(* CoDeSys 2.3.9.41 project: Lab4.pro *)
(* Libraries: STANDARD.LIB 5.6.98 11:03:02 *)

(* Task configuration *)
TASK Standard (PRIORITY := 0, INTERVAL := T#5ms);
	MAIN
END_TASK

(* Global variable list: Global_Variables *)
VAR_GLOBAL
END_VAR

VAR_GLOBAL CONSTANT
	F_TASK : INT := 200;
	PERIOD_TASK : INT := 5;
END_VAR

(* POU MAIN, ST *)
PROGRAM MAIN
VAR
	lp : LowpassFilter;
	integrate : Integrator;

END_VAR
Generator();
END_PROGRAM

(* POU LowpassFilter, ST *)
FUNCTION_BLOCK LowpassFilter
VAR_INPUT
	input : REAL;
	tau : INT;
END_VAR
VAR_OUTPUT
	output : REAL;
END_VAR
VAR
	sum : REAL := 0;
END_VAR
sum := (input * PERIOD_TASK + sum * tau) / (PERIOD_TASK + tau);
output := sum;
END_FUNCTION_BLOCK

(* POU Integrator, ST *)
FUNCTION_BLOCK Integrator
VAR_INPUT
	input : REAL;
END_VAR
VAR_OUTPUT
	output : REAL;
END_VAR
VAR
	sum : REAL := 0;
END_VAR
sum := sum + input;
output := sum;
END_FUNCTION_BLOCK

(* POU Generator, ST *)
PROGRAM Generator
VAR
	t : UINT := 0;
	a : REAL := 1;
	offset : REAL := 0;
	w : REAL := 1.0;
	duty : REAL := 0.25;
	sinus : REAL;
	square : REAL;
	pwm : REAL;
END_VAR
IF t <= REAL_TO_INT(w*F_TASK) THEN
	t := t + 1;
ELSE
	t := 0;
END_IF
sinus := SinusFunction(a, offset, w, t);
square := SquareSignal(a, offset, w, t);
pwm := PwmSignal(a, offset, w, t, duty);
END_PROGRAM

(* POU SinusFunction, ST *)
FUNCTION SinusFunction : REAL
VAR_INPUT
	a : REAL;
	offset : REAL;
	w : REAL;
	t : INT;
END_VAR
VAR
END_VAR
SinusFunction := a * SIN(INT_TO_REAL(t)*w /F_TASK *2.0*3.1415) + offset;
END_FUNCTION

(* POU SquareSignal, ST *)
FUNCTION SquareSignal : REAL
VAR_INPUT
	a : REAL;
	offset : REAL;
	w : REAL;
	t : INT;
END_VAR
VAR
	per : INT;
END_VAR
per := REAL_TO_INT(F_TASK / w);
IF (t MOD per) < (per / 2) THEN
	SquareSignal := offset + a;
ELSE
	SquareSignal := offset - a;
END_IF
END_FUNCTION

(* POU PwmSignal, ST *)
FUNCTION PwmSignal : REAL
VAR_INPUT
	a : REAL;
	offset : REAL;
	w : REAL;
	t : INT;
	duty : REAL;
END_VAR
VAR
	per : INT;
END_VAR
per := REAL_TO_INT(F_TASK / w);
IF duty*per >= per THEN
	PwmSignal := offset + a;
ELSIF duty*per <=0 THEN
	PwmSignal := offset - a;
ELSIF (t MOD per) < duty*per THEN
	PwmSignal := offset + a;
ELSE
	PwmSignal := offset - a;
END_IF
END_FUNCTION

(* POU EdgeDetector, ST *)
FUNCTION_BLOCK EdgeDetector
VAR_INPUT
	inputValue : BOOL;
END_VAR
VAR_OUTPUT
	risingEdge : BOOL;
	fallingEdge : BOOL;
END_VAR
VAR
	prev : BOOL := FALSE;
END_VAR
IF inputValue > prev THEN
	risingEdge := TRUE;
	fallingEdge := FALSE;
ELSIF inputValue < prev THEN
	risingEdge := FALSE;
	fallingEdge := TRUE;
ELSE
	risingEdge := FALSE;
	fallingEdge := FALSE;
END_IF
prev := inputValue;
END_FUNCTION_BLOCK

(* POU EdgeDetectorDouble, ST *)
FUNCTION_BLOCK EdgeDetectorDouble
VAR_INPUT
	inputValue : BOOL;
	threshold : INT;
END_VAR
VAR_OUTPUT
	risingEdge : BOOL;
	fallingEdge : BOOL;
	double : BOOL;
END_VAR
VAR
	prev : BOOL := FALSE;
	timer : INT := 0;
END_VAR
IF inputValue > prev THEN
	risingEdge := TRUE;
	fallingEdge := FALSE;
	IF timer < threshold THEN
		double := TRUE;
	ELSE
		double := FALSE;
	END_IF
	timer := 0;
ELSIF inputValue < prev THEN
	risingEdge := FALSE;
	fallingEdge := TRUE;
	IF timer < 32767 THEN
		timer := timer + 1;
	END_IF
	double := FALSE;
ELSE
	risingEdge := FALSE;
	fallingEdge := FALSE;
	IF timer < 32767 THEN
		timer := timer + 1;
	END_IF
	double := FALSE;
END_IF
prev := inputValue;
END_FUNCTION_BLOCK

(* POU SecondOrderLag, ST *)
FUNCTION_BLOCK SecondOrderLag
VAR_INPUT
	input : REAL;
	omega : REAL;
	d : REAL;
END_VAR
VAR_OUTPUT
	output : REAL;
END_VAR
VAR
	sum1 : REAL := 0;
	sum2 : REAL := 0;
END_VAR
output :=
(PERIOD_TASK * PERIOD_TASK * omega * omega * input
	+ (2 * d * PERIOD_TASK * omega + 2) * sum1
	- sum2) /
(PERIOD_TASK * omega * omega + 2 * d * PERIOD_TASK * omega + 1);
sum2 := sum1;
sum1 := output;
END_FUNCTION_BLOCK
